{attribute 'qualified_only'}
VAR_GLOBAL
	fSimulationTime : LREAL; 
	bSimulationStarted : BOOL;
	fCylinderVelocity : LREAL;
	fCylinderPosition : LREAL;
END_VAR

(* stored: Version 1.1.0.1, ProductVersion 3.1.4024.9
   GVL Outputs: Id {6100726c-2a37-4206-8249-64f2ca6ce4cf} *)
